{attribute 'qualified_only'}
VAR_GLOBAL CONSTANT 
	speedMatrixSize : UINT := 10;
	 
END_VAR

(* stored: Version 1.1.0.1, ProductVersion 3.1.4024.12
   GVL Constants: Id {c6b77bf3-a747-46fb-bd08-4e166f6eb3e6} *)
